{attribute 'linkalways'} 
{attribute 'no_explicit_call' := 'This FB is a CLASS and must be accessed using methods or properties'}
{attribute 'enable_dynamic_creation'}
FUNCTION_BLOCK _LREAL EXTENDS NumericDatatypeBase
VAR
	localData : LREAL;
	activeData : REFERENCE TO LREAL REF= localData;
END_VAR

PROPERTY PUBLIC Address : PVOID
GET
Address := ADR(activeData);
END_GET
END_PROPERTY

METHOD PUBLIC ClearReference
VAR_INPUT
END_VAR
activeData REF= localData;
END_METHOD

METHOD PUBLIC Clone : I_Datatype
VAR
    pClone : POINTER TO _LREAL;
END_VAR
pClone := __NEW(_LREAL(InitialValue := Value));
Clone := pClone^;
END_METHOD

METHOD FB_init : BOOL
VAR_INPUT
	bInitRetains : BOOL; // if TRUE, the retain variables are initialized (warm start / cold start)
	bInCopyCode : BOOL;  // if TRUE, the instance afterwards gets moved into the copy code (online change)
	InitialValue : LREAL;
END_VAR
localData := InitialValue;
END_METHOD

PROPERTY PUBLIC IsFloat : BOOL
GET
IsFloat := TRUE;
END_GET
END_PROPERTY

PROPERTY PUBLIC IsSigned : BOOL
GET
IsSigned := TRUE;
END_GET
END_PROPERTY

METHOD PUBLIC MakeReferenceTo
VAR_INPUT
	ReferenceTarget : REFERENCE TO LREAL;
END_VAR
activeData REF= ReferenceTarget;
END_METHOD

PROPERTY PUBLIC MaxValue : LREAL
GET
MaxValue :=  DatatypeLimits.LREAL_MAX_VALUE;
END_GET
END_PROPERTY

PROPERTY PUBLIC MinValue : LREAL
GET
MinValue := DatatypeLimits.LREAL_MIN_VALUE;
END_GET
END_PROPERTY

METHOD PROTECTED SerializeMaxValue
VAR_INPUT
	Serializer : I_Serializer;
END_VAR
Serializer.AddLreal(MaxValue);
END_METHOD

METHOD PROTECTED SerializeMinValue
VAR_INPUT
	Serializer : I_Serializer;
END_VAR
Serializer.AddLreal(MinValue);
END_METHOD

METHOD PUBLIC SerializeWith
VAR_INPUT
	Serializer : I_Serializer;
END_VAR
Serializer.AddLreal(activeData);
END_METHOD

PROPERTY PUBLIC Size : UDINT
GET
Size := SIZEOF(activeData);
END_GET
END_PROPERTY

METHOD TryDeserializeFrom : BOOL
VAR_INPUT
	Deserializer : I_Deserializer;
	Feedback : I_DeserializerFeedback;
END_VAR
TryDeserializeFrom := Deserializer.TryGetLreal(activeData, Feedback);
END_METHOD

METHOD TryMakeReferenceTo : BOOL
VAR_INPUT
	Target : I_Datatype;
END_VAR
VAR
	pTargetData : POINTER TO LREAL;
END_VAR
IF NOT (Target.TypeName = TypeName) THEN
	RETURN;
END_IF

pTargetData := Target.Address;
activeData REF= pTargetData^;
TryMakeReferenceTo := TRUE;
END_METHOD

PROPERTY PUBLIC TypeName : T_MAXSTRING
GET
TypeName := 'LREAL';
END_GET
END_PROPERTY

PROPERTY PUBLIC Value : LREAL
GET
Value := activeData;
END_GET
SET
activeData := Value;
END_SET
END_PROPERTY

END_FUNCTION_BLOCK

(* stored: Version 1.1.0.1, ProductVersion 3.1.4024.12
   POU _LREAL: Id {8e067bb4-51c1-03ba-0bbd-4862f2523717}, SpecialFunc None
   Folder Constructor: Id {eb3753b0-9f5f-0762-2da0-0adc70fd1a33}
   Folder Protected: Id {3c4e0835-1ab7-4a86-9ef2-35fda4f00373}
   Property Address: Id {8e03e558-4a34-07a7-06c0-57a22c8eec72}
   Get Get: Id {b699162c-7b65-0274-3a31-2f4733d1714a}
   Method ClearReference: Id {c639a08c-bafa-0038-3b8f-f2ee89a2d3b0}
   Method Clone: Id {b78988db-dc44-04c2-1c26-708f82ca0811}
   Method FB_init: Id {b3cf6c10-9e66-0036-0e9a-c3231cc8adbf}
   Property IsFloat: Id {8cd2d708-b571-0d2c-297d-fdc0590f64b0}
   Get Get: Id {b40b49fb-b78f-0c42-32ee-cbed04d379ce}
   Property IsSigned: Id {aeedeb7e-1ba0-0943-3de1-e8da8877bc20}
   Get Get: Id {ce948fe2-3d2c-0d16-1cc6-0a2b11792830}
   Method MakeReferenceTo: Id {8fdb47fb-65df-0d0d-3349-47735a971f9a}
   Property MaxValue: Id {ceb8a57c-cebb-4243-8d01-af9fc9bfc4ae}
   Get Get: Id {c9fe1856-e89b-4e85-bb49-f570ed4e6ba1}
   Property MinValue: Id {36168685-ee89-4c4f-a521-7f4d666855bc}
   Get Get: Id {95951b3d-d66f-4e3f-8051-54d229a837fd}
   Method SerializeMaxValue: Id {0796c19d-6123-4059-afd4-f2c51320b476}
   Method SerializeMinValue: Id {270e72db-be3e-409e-bc50-09dc22774e8b}
   Method SerializeWith: Id {40a92b8d-e560-0d74-0dc1-6dd2cb571dd2}
   Property Size: Id {cbc1f645-36e4-0608-3f4b-0c6b22b2e945}
   Get Get: Id {181b057c-1126-0827-2a17-64bd5d364717}
   Method TryDeserializeFrom: Id {711f7ad0-f962-000b-25c2-02854e312ae7}
   Method TryMakeReferenceTo: Id {ac5ac32b-a62f-0da1-0a6a-cd48f6969026}
   Property TypeName: Id {e6316010-6ea7-03df-1fc2-e99b11b7beb6}
   Get Get: Id {b84d9190-6f40-00d5-3d70-6d8b22c8e8c3}
   Property Value: Id {6503b810-eb6a-0f1a-0982-25f7a5b8469b}
   Get Get: Id {97728efa-957e-0010-1235-2c7994e7bc7f}
   Set Set: Id {9a159a22-9519-007c-3505-f23c162c3708} *)
